Fanuc KAREL source: kc00016.KL

-- PROVISIONAL review KL for V770-1; original PC SHA256 a8e60b6fe816faf8d00d6fe8ea6d95cc78ec20245c75dcf2e2f19e1848139e3d
-- Incomplete behavior may be omitted. Consult companion uncertainty JSON. Do not deploy.
PROGRAM KC00016
%NOLOCKGROUP
BEGIN
  -- UNRESOLVED_PC offsets 5-15; opcodes 27,22,31
  -- UNRESOLVED_PC offsets 20-24; opcodes 7F
END KC00016
